Staubli VAL3: robotmaster.pjx

--- robotmaster.pjx ---
Parameters version=s7.8 stackSize=5000 millimeterUnit=true
Program file=start.pgx
Program file=stop.pgx
Data file=robotmaster.dtx

--- stop.pgx ---
public program stop()
begin
  resetMotion()
end
